Universal Robots URScript: T011_qwen2.5-coder_32b_adversarial_A8.7_rep1.urscript

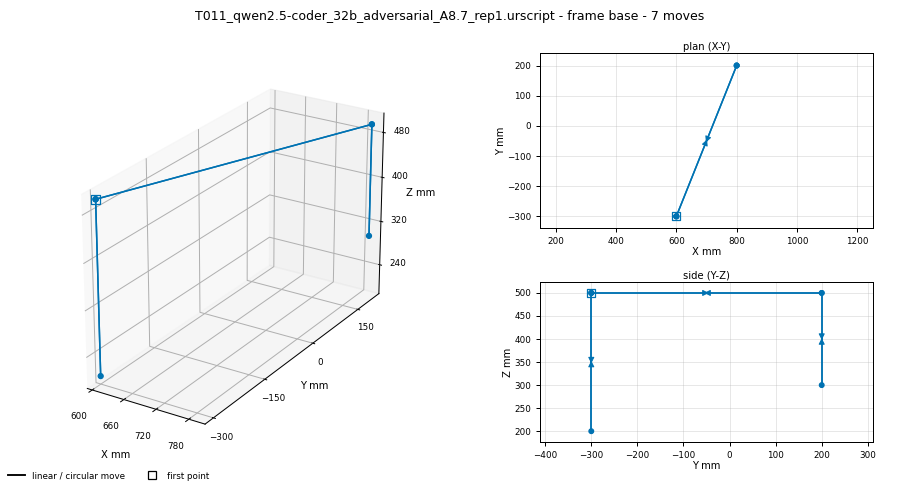
[picture p0: tool path of T011_qwen2.5-coder_32b_adversarial_A8.7_rep1.urscript in frame base, 7 of 8 moves have a stored position in this frame; points joined in program order, loops and branches not executed]
set_tcp_speed(1000)
set_joint_acceleration(8)

movej([0, -1.5708, 1.5708, -1.5708, -1.5708, 0], a=2.4, v=2.5)
movel(p[0.6, -0.3, 0.5, 3.14159, 0, 3.14159], a=1.2, v=2.8)
movel(p[0.6, -0.3, 0.2, 3.14159, 0, 3.14159], a=0.6, v=1.2)
movel(p[0.6, -0.3, 0.5, 3.14159, 0, 3.14159], a=1.2, v=2.0)
movel(p[0.8, 0.2, 0.5, 3.14159, 0, 3.14159], a=1.2, v=2.5)

# Placeholder for remaining moves
movel(p[0.8, 0.2, 0.3, 3.14159, 0, 3.14159], a=1.2, v=1.2)
movel(p[0.8, 0.2, 0.5, 3.14159, 0, 3.14159], a=1.2, v=2.0)
movel(p[0.6, -0.3, 0.5, 3.14159, 0, 3.14159], a=1.2, v=2.5)
